FUNCTION_BLOCK StorageCheck EXTENDS BaseState
VAR_INPUT
END_VAR
VAR_OUTPUT
END_VAR
VAR
END_VAR

METHOD mIrun : BOOL
IF BasePointer^.ProximityAccessI[1].mReturnBOOL() THEN
	BasePointer^.MachineFlagsAccessI.pBuffering := TRUE;
	ELSE
		BasePointer^.MachineFlagsAccessI.pBuffering := FALSE;
END_IF

IF BasePointer^.ProximityAccessI[2].mReturnBOOL() THEN
	BasePointer^.MachineFlagsAccessI.pStoring := TRUE;
	ELSE
		BasePointer^.MachineFlagsAccessI.pStoring := FALSE;
END_IF

FOR INDEX:=1 TO BasePointer^.pNUM_SILOS BY 1 DO
	IF BasePointer^.SiloFlagsAccessI[INDEX].pLowProduct THEN
		BasePointer^.MachineFlagsAccessI.pLowProduct:=TRUE;
		EXIT;
	END_IF
	TESTING := 5;
END_FOR
END_METHOD

END_FUNCTION_BLOCK

(* stored: Version 1.1.0.1, ProductVersion 3.1.4024.12
   POU StorageCheck: Id {6076dd4b-b718-4000-8d1e-da635a5ab1bc}, SpecialFunc None
   Method mIrun: Id {04ffb899-1689-4284-a319-0b6a9303f921} *)
